TYPE T_DB_LongSTRING : STRING(1024);
END_TYPE

(* stored: Version 1.1.0.1, ProductVersion 3.1.4024.15
   DUT T_DB_LongSTRING: Id {d0deb71a-2bed-4b99-8155-544e8b3dd332} *)
